RoboDK station: Industrial.rdk

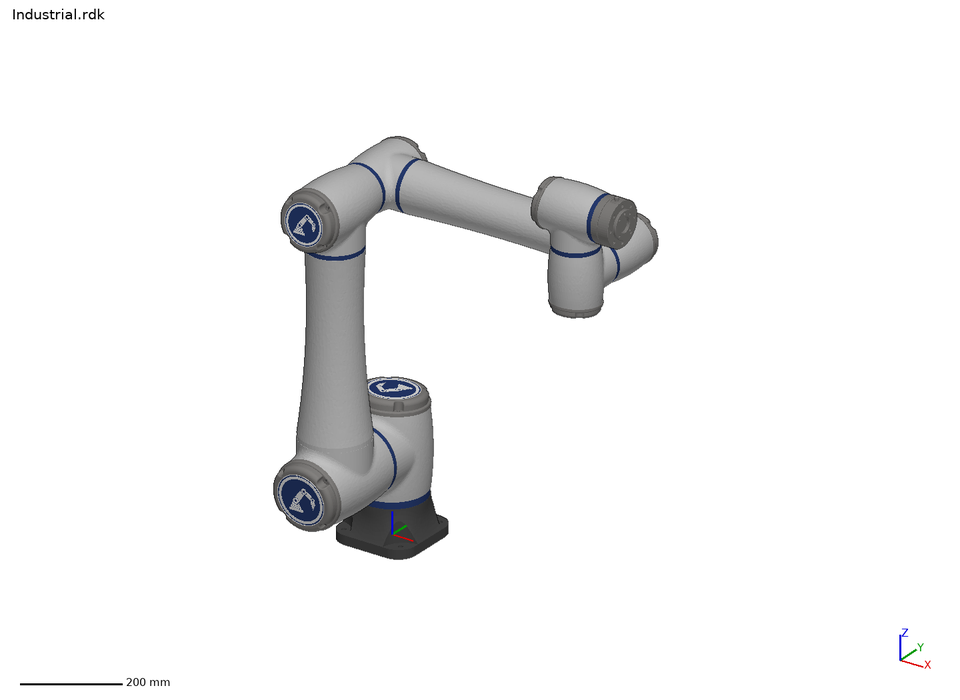
[picture v0: the station drawn from its stored meshes, robots at their saved joint values, targets as dots, program paths as lines]
Station Industrial (saved by RoboDK 6.0.1). Poses are relative to the parent item; angles as X-Y-Z fixed-axis rotations.
  - Python program Prog1 (listed below)
  - frame RoboDK RDK-COBOT-1200 Base at (0, 2000, 0) mm
    - robot RoboDK RDK-COBOT-1200: 6 axes
        modified DH rows (alpha deg, a mm, theta deg, d mm): 0, 0, 0, 201; 90, 0, 90, 0; 0, 590, 0, 0; 0, 560, -90, 175; -90, 0, 0, 140; 90, 0, -90, 117
        joint limits [-360, -180, -160, -180, -180, -360] to [360, 180, 160, 180, 180, 360]; home [0, 0, -90, 90, 90, 0]; saved at [0, 0, -90, 90, 90, 0]

--- Python program Prog1 ---
# Type help("robodk.robolink") or help("robodk.robomath") for more information
# Press F5 to run the script
# Documentation: https://robodk.com/doc/en/RoboDK-API.html
# Reference:     https://robodk.com/doc/en/PythonAPI/robodk.html
# Note: It is not required to keep a copy of this file, your Python script is saved with your RDK project

# You can also use the new version of the API:
from robodk import robolink    # RoboDK API
from robodk import robomath    # Robot toolbox
RDK = robolink.Robolink()

# Forward and backwards compatible use of the RoboDK API:
# Remove these 2 lines to follow python programming guidelines
from robodk import *      # RoboDK API
from robolink import *    # Robot toolbox
# Link to RoboDK
# RDK = Robolink()

# Notify user:
print('To edit this program:\nright click on the Python program, then, select "Edit Python script"')

# Program example:
item = RDK.Item('base')
if item.Valid():
    print('Item selected: ' + item.Name())
    print('Item posistion: ' + repr(item.Pose()))

print('Items in the station:')
itemlist = RDK.ItemList()
print(itemlist)

# Provoking an exception will display the console output if you run this script from RoboDK
raise Exception('Program not edited.')
